// SIMATIC S7-200 project (STEP 7-Micro/WIN), CPU 224 REL 01.22

ORGANIZATION_BLOCK MAIN:OB1
TITLE=【恒压供水控制系统（三）】
// 这是我写的第三个恒压供水系统，、支持手动/自动切换、PID压力控制、三台主泵和一台备用泵的轮换运行以及故障切换功能。
// 系统涉及三台主泵、一台备用泵、变频器、压力传感器、手动/自动切换按钮、系统报警指示灯、水泵故障指示灯、系统运行指示灯和PID运行指示灯。
// 系统通过手动/自动切换按钮实现运行模式的切换，由自动模式标志决定。操作员按下系统启动按钮启动系统，按下系统停止按钮停止系统。
// 在自动模式下，系统启动后，依靠压力传感器输入实时监测水压，并通过PID压力控制功能调整变频器频率输出，维持恒压。变频器启动信号置位后，频率输出由最低和最高频率标志监控。
// 系统管理三台主泵，通过变频接触器控制，每隔约1小时轮换运行，确保均衡使用。系统通过轮换逻辑确保同一时刻通常只有一台主泵变频运行。
// 例如，当一台主泵变频运行时，若变频器频率达到最高，主泵工频接触器通过延时启动，但应避免与变频接触器同时运行。若主泵故障，系统置位故障标志，并通过故障切换标志启动备用泵工频接触器。备用泵运行时，应确保与主泵工频接触器不同时运行，但当前实现可能允许同时运行。若需高效运行，可通过备用泵变频启动脉冲启动备用泵变频接触器。
// 此外，当系统检测到所有主泵和备用泵停止时，设置辅助泵待启标志。当辅助泵待启标志置位，且PID输出显示压力不足时，辅助泵启动信号通过延时置位，避免压力正常时误启。若变频器频率达到最高，辅助泵随后停止运行。
// 
// 
BEGIN
Network 1 // Network Title
// 初始化调用子程序0
LD     SM0.1
CALL   SBR_0:SBR0, VD0
?000
Network 2
// 手动/自动转换
LD     I0.0
LPS
TON    T37, +10
A      T37
A      I0.1
EU
S      M0.0, 1
LPP
A      I0.2
R      M0.0, 1
Network 3
// 每隔4小时轮流交替倒泵延时时间
LD     SM0.0
LPS
A      Q0.2
AN     Q0.3
AN     Q0.5
AN     T44
TON    T44, +3600
LRD
A      Q0.4
AN     Q0.1
AN     Q0.5
AN     T45
TON    T45, +3600
LRD
A      Q0.6
AN     Q0.1
AN     Q0.3
AN     T46
TON    T46, +3600
LRD
A      Q1.1
TON    T50, +18000
LRD
A      T50
S      M4.3, 1
LPP
A      SM0.1
R      M4.3, 1
Network 4
LD     SM0.0
A      T44
LD     T47
O      SM0.1
CTU    C0, VW8
Network 5
LD     SM0.0
A      T45
LD     T48
O      SM0.1
CTU    C1, VW8
Network 6
LD     SM0.0
A      T46
LD     T49
O      SM0.1
CTU    C2, VW8
Network 7
LD     C0
O      C1
O      C2
O      T50
O      T53
EU
=      M4.2
Network 8
// 变频器最低和最高频率输出上升沿脉冲
LD     M0.0
LPS
AR<=   VD108, 0.2
TON    T38, +10
A      T38
EU
S      M5.0, 1
LPP
AR>=   VD108, 0.7
TON    T39, 500
A      T39
EU
=      M5.1
Network 9
LD     M0.6
O      M1.2
O      M1.5
O      M2.5
O      M2.6
O      M2.7
R      M5.0, 1
Network 10
// 1#泵变频接触器启动
LD     M0.0
LPS
EU
=      M0.1
LRD
LD     M0.1
LDN    M1.6
A      T98
OLD
O      T42
O      Q0.2
ALD
AN     T34
AN     T100
=      Q0.2
LPP
TON    T33, +5
Network 11
// 延时50ms后变频器启动。
LD     M0.0
LPS
A      T33
AN     M0.2
=      Q0.0
LRD
LD     M5.1
O      M3.7
O      M4.2
ALD
EU
S      M0.2, 1
LPP
LD     T35
O      T97
O      T99
O      T41
O      T43
O      T47
O      T48
O      T49
O      T52
O      T55
ALD
EU
R      M0.2, 1
Network 12
// 从1#泵变频切换到2#泵变频的时间延时
LD     M0.0
LPS
LD     M5.1
O      C0
LD     Q0.2
LD     I0.5
A      Q1.0
OLD
ALD
ALD
EU
S      M0.3, 1
LRD
LD     Q0.1
O      T47
ALD
EU
R      M0.3, 1
LRD
A      M0.3
TON    T34, +10
LPP
A      T34
LPS
AN     C0
TON    T35, +10
LPP
A      C0
TON    T47, +10
Network 13
// 2#泵变频接触器启动
LD     M0.0
LPS
A      T34
AN     I0.6
EU
=      M0.4
LPP
LD     M0.4
O      Q0.4
ALD
AN     T36
AN     T100
=      Q0.4
Network 14
// 1#泵工频接触器启动和停止
LD     M0.0
LPS
A      T35
EU
=      M0.5
LRD
LD     M0.5
O      Q0.1
ALD
AN     I0.5
AN     M0.6
=      Q0.1
LPP
A      M5.0
LDN    I0.6
AN     I0.7
AN     Q0.5
LD     Q0.4
O      Q0.6
ALD
LD     I0.6
AN     Q0.5
LD     Q1.0
O      Q0.6
ALD
OLD
LD     I0.7
AN     Q0.7
LD     Q0.4
O      Q1.0
ALD
OLD
ALD
=      M0.6
Network 15
// 从2#泵变频切换到3#泵变频的时间延时
LD     M0.0
LPS
LD     M5.1
O      C1
LD     Q0.4
LD     I0.6
A      Q1.0
OLD
ALD
ALD
EU
S      M0.7, 1
LRD
LD     Q0.3
O      T48
ALD
EU
R      M0.7, 1
LRD
A      M0.7
TON    T36, +10
LPP
A      T36
LPS
AN     C1
TON    T97, +10
LPP
A      C1
TON    T48, +10
Network 16
// 3#泵变频接触器启动
LD     M0.0
LPS
A      T36
AN     I0.7
EU
=      M1.0
LPP
LD     M1.0
O      Q0.6
ALD
AN     T98
AN     T100
=      Q0.6
Network 17
// 2#泵工频接触器启动和停止
LD     M0.0
LPS
A      T97
EU
=      M1.1
LRD
LD     M1.1
O      Q0.3
ALD
AN     I0.6
AN     M1.2
=      Q0.3
LPP
A      M5.0
LDN    I0.5
AN     I0.7
AN     Q0.1
LD     Q0.2
O      Q0.6
ALD
LD     I0.5
AN     Q0.7
LD     Q1.0
O      Q0.6
ALD
OLD
LD     I0.7
AN     Q0.1
LD     Q0.2
O      Q1.0
ALD
OLD
ALD
=      M1.2
Network 18
LD     Q0.1
A      Q0.3
A      Q0.6
LD     Q0.3
A      Q0.5
A      Q0.2
OLD
LD     Q0.5
A      Q0.1
A      Q0.4
OLD
=      M5.2
Network 19
// 从3#泵变频切换到1#泵变频的时间延时(当1#泵发生故障时，切换到备用泵变频）
LD     M0.0
LPS
LD     M5.1
O      C2
AN     M5.2
LD     Q0.6
LD     I0.7
A      Q1.0
OLD
ALD
ALD
EU
S      M1.3, 1
LRD
LD     Q0.5
O      T49
ALD
EU
R      M1.3, 1
LRD
A      M1.3
TON    T98, +10
LPP
A      T98
LPS
AN     C2
TON    T99, +10
LPP
A      C2
TON    T49, +10
Network 20
// 3#泵工频接触器启动和停止
LD     M0.0
LPS
A      T99
AN     I0.7
EU
=      M1.4
LRD
LD     M1.4
O      Q0.5
ALD
AN     I0.7
AN     M1.5
=      Q0.5
LPP
A      M5.0
LDN    I0.5
AN     I0.6
AN     Q0.3
LD     Q0.2
O      Q0.4
ALD
LD     I0.5
AN     Q0.3
LD     Q1.0
O      Q0.4
ALD
OLD
LD     I0.6
AN     Q0.7
LD     Q0.2
O      Q1.0
ALD
OLD
ALD
=      M1.5
Network 21
// 1#泵发生故障
LD     M0.0
LPS
A      I0.5
LPS
A      Q0.1
S      M1.6, 1
LRD
A      M1.6
EU
=      M1.7
LPP
LD     M1.7
O      T35
ALD
=      M2.0
LPP
AN     I0.5
R      M1.6, 1
Network 22
// 2#泵发生故障
LD     M0.0
A      I0.6
LPS
A      Q0.3
EU
=      M2.1
LPP
LD     M2.1
O      T97
ALD
=      M2.2
Network 23
// 3#泵发生故障
LD     M0.0
A      I0.7
LPS
A      Q0.5
EU
=      M2.3
LPP
LD     M2.3
O      T99
ALD
=      M2.4
Network 24
// 当1#、2#、3#泵发生故障时，备用泵投入运行，备用泵工频接触器启动
LD     M0.0
LD     I0.5
O      I0.6
O      I0.7
ALD
LPS
LD     M2.0
O      M2.2
O      M2.4
O      Q0.7
ALD
AN     M2.5
AN     M2.6
AN     M2.7
=      Q0.7
LRD
A      I0.5
A      M5.0
AN     Q0.5
LD     Q0.4
O      Q0.6
ALD
=      M2.5
LRD
A      I0.6
A      M5.0
AN     Q0.1
LD     Q0.6
O      Q0.2
ALD
=      M2.6
LPP
A      I0.7
A      M5.0
AN     Q0.3
LD     Q0.2
O      Q0.4
ALD
=      M2.7
Network 25
// 在发生故障期间，从1#、2#、3#泵切换到备用泵变频接触器
LD     M0.0
LPS
A      I0.5
LPS
A      T98
EU
=      M3.0
LPP
LD     M3.0
O      M3.1
ALD
AN     T34
AN     T100
=      M3.1
LRD
A      I0.6
LPS
A      T34
EU
=      M3.2
LPP
LD     M3.2
O      M3.3
ALD
AN     T36
AN     T100
=      M3.3
LPP
A      I0.7
LPS
A      T36
EU
=      M3.4
LPP
LD     M3.4
O      M3.5
ALD
AN     T98
AN     T100
=      M3.5
Network 26
// 备用泵变频接触器启动
LD     SM0.0
LPS
LD     M3.1
O      M3.3
O      M3.5
O      M4.4
ALD
=      Q1.0
LRD
LPS
A      T51
EU
S      M4.4, 2
LRD
A      M4.5
TON    T52, +10
LRD
A      T52
R      M4.5, 1
LRD
A      M4.4
TON    T53, +600
LPP
A      T53
TON    T54, +10
LRD
A      T54
R      M4.4, 1
S      M4.6, 1
LPP
LPS
A      M4.6
TON    T55, +10
LRD
A      T55
R      M4.6, 1
LPP
A      SM0.1
R      M4.4, 3
Network 27
// 辅助泵变频启动
LD     M0.0
LPS
AN     Q0.1
AN     Q0.3
AN     Q0.5
AN     Q0.7
=      M3.6
LRD
A      M3.6
A      Q0.0
AR<=   VD108, 0.2
AN     T41
TON    T40, +50
LRD
A      T40
EU
=      M3.7
LRD
LD     M3.7
O      M4.0
ALD
LPS
AN     T100
=      M4.0
LPP
TON    T100, +80
LPP
LD     T100
O      T54
O      Q1.1
ALD
LPS
AN     T42
AN     T51
=      Q1.1
LPP
TON    T41, +1
Network 28
// 辅助泵停止
LD     M0.0
LPS
A      Q1.1
A      M5.1
S      M4.1, 1
LRD
A      M4.1
TON    T42, +1
LRD
A      M4.3
TON    T51, +10
LRD
LD     T42
O      T51
ALD
TON    T43, +1
LPP
A      T43
R      M4.1, 3
END_ORGANIZATION_BLOCK

SUBROUTINE_BLOCK SBR_0:SBR0
TITLE=POU Comment
VAR_INPUT
AI_IN:REAL;	// LD0 
END_VAR
BEGIN
Network 1 // Network Title
// 装载PID参数，连接PID中断服务程序
LD     SM0.0
MOVR   #AI_IN:LD0, VD104
MOVR   3.0, VD112
MOVR   0.5, VD116
MOVR   0.5, VD120
MOVR   0.0, VD124
MOVB   100, SMB34
ATCH   INT_0:INT0, 10
ENI
END_SUBROUTINE_BLOCK

INTERRUPT_BLOCK INT_0:INT0
TITLE=POU Comment
BEGIN
Network 1 // Network Title
// 过程变量的输入及标准化转换
LD     SM0.0
ITD    AIW0, AC0
DTR    AC0, AC0
/R     32000.0, AC0
MOVR   AC0, VD100
Network 2
// 执行PID运算
LD     SM0.0
PID    VB100, 0
Network 3
// PID运算输出及标准化转换
LD     SM0.0
MOVR   VD108, AC0
*R     32000.0, AC0
ROUND  AC0, AC0
DTI    AC0, AC0
MOVW   AC0, AQW0
MOVW   AC0, AC1
/I     +640, AC1
END_INTERRUPT_BLOCK

DATA_BLOCK_TAB USER1
BEGIN
//DATA BLOCK COMMENTS
//Press F1 for help and example data block
VD0      0.75                //压力设定
VW8      40                  //主泵轮流交替循环时间
END_DATA_BLOCK_TAB
